(* IEC 61131-3 sources: CodesysTest/export/UN00 - Sharp Bagger/EM01 - Bagger Head/CM00 - Bag Open Fingers/Base/FB_BaseBagOpenFingers.pou, 1 file *)

(* ---- FB_BaseBagOpenFingers.pou.st ---- *)
(*#-#-#-#-#-#-#-#-#-#---Declaration---#-#-#-#-#-#-#-#-#-#-#-#-#*)

FUNCTION_BLOCK FB_BaseBagOpenFingers EXTENDS FB_BaseComponent IMPLEMENTS IBagOpenFingers
VAR_INPUT
	delayToGrabSetting : REAL;						// How long to wait afer a grab request to start moving fingers
	delayToCheckBagPresentSetting : REAL;			// How long to wait after grabbing bag to check if it is present
	delayToClearSetting : REAL;						// How long to wait after letting go of bag to call it clear of the pressure bar
END_VAR
VAR_OUTPUT
	grabCounter : FB_MachineCounter(name := CONCAT(_prefix, 'Grab Counter'));
	releaseCounter : FB_MachineCounter(name := CONCAT(_prefix, 'Release Counter'));
	missedCounter : FB_MachineCounter(name := CONCAT(_prefix, 'Missed Counter'));
END_VAR
VAR
	_grabBagRequest : BOOL;
	_releaseBagRequest : BOOL;
	_bagCleared : BOOL;
	_bagGrabbed : BOOL;
	_bagMissed : BOOL;
	delayToGrab : Standard.TON;
	delayToCheckBagPresent : Standard.TON;
	delayToClear : Standard.TON;
END_VAR
VAR_IN_OUT

END_VAR(*#-#-#-#-#-#-#-#-#-#---Implementation---#-#-#-#-#-#-#-#-#-#-#-#-#*)

SUPER^();
delayToGrab(IN := _grabBagRequest, PT := REAL_TO_TIME(delayToGrabSetting * 1000));
delayToCheckBagPresent(IN := delayToGrab.Q, PT := REAL_TO_TIME(delayToCheckBagPresentSetting * 1000));
delayToClear(IN := _releaseBagRequest, PT := REAL_TO_TIME(delayToClearSetting * 1000));
